FUNCTION_BLOCK ObserveStamp EXTENDS HardwareObservationBase
VAR_INPUT
END_VAR
VAR_OUTPUT
END_VAR
VAR
	m_ptrStamp: POINTER TO Stamp;
	m_ptrStampWP: POINTER TO xPPUProduct;
	m_detectionStep: INT := 0;
END_VAR

METHOD FB_init : BOOL
VAR_INPUT
	bInitRetains : BOOL; // if TRUE, the retain variables are initialized (warm start / cold start)
	bInCopyCode : BOOL;  // if TRUE, the instance afterwards gets moved into the copy code (online change)

	i_ptrStamp: POINTER TO Stamp;
	i_ptrWP: POINTER TO xPPUProduct;
END_VAR
m_ptrStamp := i_ptrStamp;
m_ptrStampWP := i_ptrWP;
END_METHOD

METHOD  ResetDefinition : BOOL
VAR_INPUT
END_VAR
;
END_METHOD

(* Update an instance of ProcessState with the part of the process that can be observed by this Hardware Interface. *)
METHOD UpdateProcessObservation : BOOL
VAR_IN_OUT
	io_processState: ProcessState;
END_VAR
io_processState.UpdateState_Binary(EProcessVariables.Stamp_StamperExtended, m_ptrStamp^.m_stampingCylinder.Extended, i_force := TRUE);
io_processState.UpdateState_Binary(EProcessVariables.Stamp_StamperRetracted, m_ptrStamp^.m_stampingCylinder.Retracted, i_force := TRUE);
io_processState.UpdateState_Binary(EProcessVariables.Stamp_SliderExtended, m_ptrStamp^.m_slidingCylinder.Extended, i_force := TRUE);
io_processState.UpdateState_Binary(EProcessVariables.Stamp_SliderRetracted, m_ptrStamp^.m_slidingCylinder.Retracted, i_force := TRUE);

io_processState.UpdateState_Binary(EProcessVariables.Stamp_WPAtStamp, m_ptrStamp^.WPAtStart, i_force := TRUE);
m_ptrStampWP^.IsPresent := m_ptrStamp^.WPAtStart;

CASE m_detectionStep OF
	0: // initial, empty state
	io_processState.UpdateState_Numeric(EProcessVariables.Stamp_WorkpieceState, EStampStates.none, i_force := TRUE);
	m_ptrStampWP^.IsStamped := FALSE;
	IF m_ptrStamp^.WPAtStart THEN
		m_detectionStep := 1;
	END_IF
	
	1: // WP received
	io_processState.UpdateState_Numeric(EProcessVariables.Stamp_WorkpieceState, EStampStates.unpressed, i_force := TRUE);
	IF NOT m_ptrStamp^.m_slidingCylinder.Extended THEN
		m_detectionStep := 2;
	ELSIF NOT m_ptrStamp^.WPAtStart THEN
		// WP removed without stamping
		m_detectionStep := 0;
	END_IF
	
	2: // busy
	io_processState.UpdateState_Numeric(EProcessVariables.Stamp_WorkpieceState, EStampStates.busy, i_force := TRUE);
	IF m_ptrStamp^.m_slidingCylinder.Extended THEN
		m_detectionStep := 3;
	END_IF
	
	3: // finished processing
	io_processState.UpdateState_Numeric(EProcessVariables.Stamp_WorkpieceState, EStampStates.pressed, i_force := TRUE);
	m_ptrStampWP^.IsStamped := TRUE;
	IF NOT m_ptrStamp^.WPAtStart THEN
		m_detectionStep := 0;
	END_IF
	
END_CASE

io_processState.UpdateState_Defined(EProcessVariables.Stamp_WPAtStamp, TRUE);
io_processState.UpdateState_Defined(EProcessVariables.Stamp_WorkpieceState, TRUE);
io_processState.UpdateState_Defined(EProcessVariables.Stamp_StamperExtended, TRUE);
io_processState.UpdateState_Defined(EProcessVariables.Stamp_StamperRetracted, TRUE);
io_processState.UpdateState_Defined(EProcessVariables.Stamp_SliderExtended, TRUE);
io_processState.UpdateState_Defined(EProcessVariables.Stamp_SliderRetracted, TRUE);
END_METHOD

END_FUNCTION_BLOCK

(* stored: Version 1.1.0.1
   POU ObserveStamp: Id {d55b2e03-acae-47de-8cb3-e6e12e8387bd}, SpecialFunc None
   Method FB_init: Id {8e934f01-af51-4fdb-96db-49498013b4dc}
   Method ResetDefinition: Id {eeab708f-eb2a-4648-a235-8af1711a625e}
   Method UpdateProcessObservation: Id {8e60c9d8-4390-43a1-b4cd-bb578fb7e32c} *)
